// TIA Portal project "Es02_TIMER" (V18)

(* hardware
DEVICE "S71500/ET200MP station_1"  S7-1500 station
   slot 0: "Telaio di montaggio_0"  Rack  6ES7 590-1***0-0AA0
   slot 1: "PLC_1"  CPU 1516-3 PN/DP  6ES7 516-3AN01-0AB0  V2.5
      slot 3: "Display CPU_1"  6ES7591-1BA00-0AA0
   slot 2: "DI 32x24VDC HF_1"  DI 32x24VDC HF  6ES7 521-1BL00-0AB0  V2.1
   slot 3: "DQ 32x24VDC/0.5A HF_1"  DQ 32x24VDC/0.5A HF  6ES7 522-1BL01-0AB0  V1.0
   slot 4: "AI 8xU/I/RTD/TC ST_1"  AI 8xU/I/RTD/TC ST  6ES7 531-7KF00-0AB0  V2.1
   slot 5: "AQ 4xU/I ST_1"  AQ 4xU/I ST  6ES7 532-5HD00-0AB0  V2.1
*)

// ===== PLC "PLC_1"  CPU 1516-3 PN/DP =====

VAR_GLOBAL   // PLC tag table "Tabella delle variabili standard"
   "Led1" AT %Q3.0 : Bool;
   "Led2" AT %Q3.1 : Bool;
END_VAR

DATA_BLOCK "DB_Comandi"   // DB1
{ S7_Optimized_Access := 'TRUE' }
VERSION : 0.1
   VAR
      btnStart : Bool;
      btnStop : Bool;
   END_VAR
BEGIN
END_DATA_BLOCK

DATA_BLOCK "DB_Variabili"   // DB2
{ S7_Optimized_Access := 'TRUE' }
VERSION : 0.1
   VAR
      Led1 : Bool;
      Led2 : Bool;
      TimerLampeggioSTART : Bool;
      TimerLampeggioDONE : Bool;
      TimerLampeggioOUTPUT : Time;
      TimerLampeggioDURATA : Time;
      InEsecuzione : Bool;
   END_VAR
BEGIN
END_DATA_BLOCK

// folder: System blocks/Program resources

DATA_BLOCK "TimerLampeggio"   // DB3
{ S7_Optimized_Access := 'TRUE' }
AUTHOR : Simatic
FAMILY : IEC
NAME : IEC_TMR
VERSION : 1.0
// stored: InstanceOfName IEC_TIMER
"IEC_TIMER"
BEGIN
END_DATA_BLOCK

// folder: (top level)

FUNCTION "FC_Grafcet" : Void   // FC1, SCL
{ S7_Optimized_Access := 'TRUE' }
VERSION : 0.1
BEGIN
   //se premo start avvio il timer
   //
   IF "DB_Comandi".btnStart = TRUE THEN
       "DB_Variabili".InEsecuzione := TRUE;
       "DB_Comandi".btnStart := FALSE;
   END_IF;
   //se premo stop avvio il timer
   //
   IF "DB_Comandi".btnStop = TRUE THEN
       "DB_Variabili".InEsecuzione := FALSE;
       "DB_Comandi".btnStop := FALSE;
   END_IF;
   //
   //il funzionamento del timer dipende dal timer della variabile InEsecuzione e nn da 2 btn
   //
   IF "DB_Variabili".InEsecuzione = TRUE THEN
       "DB_Variabili".TimerLampeggioSTART := TRUE; //il timer inizia a contare
   ELSE
       "DB_Variabili".TimerLampeggioSTART := FALSE;
   END_IF;
   //
   //gestisco il DONE del timer (ha contato l'intervallo di tempo impostato)
   //
   IF "DB_Variabili".TimerLampeggioDONE = TRUE AND "DB_Variabili".InEsecuzione = TRUE THEN
       // il timer ha contato fino alla fine
       // e voglio riprendere il ciclo dall'inizio
       "DB_Variabili".TimerLampeggioDONE := FALSE;
       "DB_Variabili".TimerLampeggioSTART := FALSE;
       //accendo-spengo le uscite
       "DB_Variabili".Led1 := NOT "DB_Variabili".Led1;
       "DB_Variabili".Led2 := NOT "DB_Variabili".Led2;
   END_IF;
END_FUNCTION

FUNCTION "FC_Timer" : Void   // FC2, SCL
{ S7_Optimized_Access := 'TRUE' }
VERSION : 0.1
BEGIN
   //imposto la durata del timer
   "DB_Variabili".TimerLampeggioDURATA := T#5s;
   "TimerLampeggio".TON(IN:="DB_Variabili".TimerLampeggioSTART,
                        PT:="DB_Variabili".TimerLampeggioDURATA,
                        Q=>"DB_Variabili".TimerLampeggioDONE,
                        ET=>"DB_Variabili".TimerLampeggioOUTPUT);
END_FUNCTION

FUNCTION "FC_Uscite" : Void   // FC3, SCL
{ S7_Optimized_Access := 'TRUE' }
VERSION : 0.1
BEGIN
   //scrivo fisicamente le uscite, dopo aver controllato che tutte le condizioni siano verificate
   //
   //IF apricancello = TRUE AND fotocellula = FALSE THEN
   //    "Led1" := TRUE
   //END_IF
   "Led1" := "DB_Variabili".Led1;
   "Led2" := "DB_Variabili".Led2;
END_FUNCTION

ORGANIZATION_BLOCK "Main"   // OB1, LAD, ProgramCycle
TITLE = "Main Program Sweep (Cycle)"
{ S7_Optimized_Access := 'TRUE' }
VERSION : 0.1
   VAR_INPUT
      Initial_Call : Bool;   // Initial call of this OB
      Remanence : Bool;   // =True, if remanent data are available
   END_VAR
   VAR_TEMP   // added for the SCL form of the ladder/FBD networks
      _w1 : Bool;
      _w2 : Bool;
   END_VAR
BEGIN

REGION Network 1
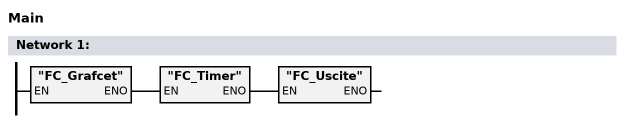
   RUNG wire#powerrail
      "FC_Grafcet"()
      "FC_Timer"()
      "FC_Uscite"()
   END_RUNG
   // the same network as SCL:
   "FC_Grafcet"(ENO => #_w1);
   "FC_Timer"(EN := #_w1, ENO => #_w2);
   IF #_w2 THEN "FC_Uscite"(); END_IF;
END_REGION
END_ORGANIZATION_BLOCK